{attribute 'reflection'}
{attribute 'hide_all_locals'}
FUNCTION_BLOCK Mover IMPLEMENTS iMover;

VAR_INPUT
	
	MotionParameters		: MotionParameters_typ;		// Motion parameters used by internal motion function blocks
	SourceInstancePath		: STRING	:= 'Direct access';					// Used internally to temporarily store the source of a Mover method call for logging purposes. Don't read or write

END_VAR
VAR_OUTPUT
	
	Ready			: BOOL;			// Mover is enabled and ready to accept motion commands
	Busy			: BOOL;			// Mover is processing a command or changing state
	
	Error			: BOOL;			// error is currently active
	ErrorID			: UDINT;		// errorID of the active error
	ErrorOrigin		: STRING;		// error source, in case of errored internal function block
	
	InGroup			: BOOL;			// Mover is currently grouped for CA
	IdentInGroup	: UDINT;		// IDX within group, for knowing which movers are adjacent
	
	AxisReference	: AXIS_REF;		// Motion link variable. Left as output so the link can be made directly, and accessed by external code
	
	TrackInfo		: TrackInfo;	// Track information as read from MC_ReadTrackPositions

END_VAR
VAR

	{attribute 'instance-path'}
	{attribute 'noinit'}
	{attribute 'hide'}
	InstancePath		: STRING;	// instance naming, for diagnostics purposes
	
	internalEnable		: BOOL;		// moves the axis from Disabled to Standstill, adds Axis to CA group, and triggers M1 Detection if configured
	internalDisable		: BOOL;		// moves the axis from Standstill to Disabled, removes Axis from CA Group
	
	internalCurrentMoveType			: MoverCommandType_enum;	// Most recent move command type
	internalReissue					: BOOL;						// reissue last command flag alows summing of all reissue commands per-scan
	
	internalCurrentDestPosition		: LREAL;						// Track position of the current motion destination;
	internalCurrentDestObjective	: STRING;						// Instance path of the current destination objective
	internalCurrentDestStation		: REFERENCE TO Station;			// Reference to a destination station, if that is the current movetype
	internalCurrentDestMultiStation	: REFERENCE TO MultiStation;	// Reference to a destination station, if that is the current movetype

	internalState			: MoverState_enum;		// Internal state variable
	internalTrackState		: TrackState;			// Internal state variable for track
	internalTrackStateDelay : TON;					// Internal timer for activate track delay
	
	internalMasterMover				: REFERENCE TO Mover;	// Internal reference to a target master mover
	internalMasterAxis				: REFERENCE TO AXIS_REF;	// Internal reference to a target master external axis
	internalGap						: LREAL;	// Gap distance to master mover during sync
	
	// Configurable Payload description	
	internalPayload			: Payload_typ;	// E.g. 0: No Product, 1: Product Loaded, 2: Product Reject. Can be modified for application
	
	// Track management
	internalTrack			: POINTER TO Track;	// Internal current track
	internalTrackIsReady	: BOOL := TRUE;			// track is ready for commands (off when .ActivateTrack is working)
	internalActivatingTrack : POINTER TO Track;	// while NOT .internalTrackIsReady the in-transition-to track is held here
	internalActivateTrackFlag	: BOOL;				// activate track requested
	
	// Internal function blocks	
	fbPower					: MC_Power;
	fbReset					: MC_Reset;
	fbStop					: MC_Stop;
	
	fbHaltCA				: MC_HaltCA;

	fbMoveAbsCA				: ARRAY[0..1] OF MC_MoveAbsoluteCA;
	fbAddToGroup			: MC_AddAxisToGroup;
	fbRemoveFromGroup		: MC_RemoveAxisFromGroup;
	
	fbGearInPosAxisCA		: ARRAY[0..1] OF MC_GearInPosCA;
	fbGearInPosMoverCA		: ARRAY[0..1] OF MC_GearInPosCA;
	
	fbGroupStatus			: MC_GroupReadStatus;
	fbGroupEnable			: MC_GroupEnable;
	fbGroupReset			: MC_GroupReset;
	fbGroupStop				: MC_GroupStop;
	
	fbReadStatus			: MC_ReadStatus;
	fbMoveRelCA				: ARRAY[0..1] OF MC_MoveRelativeCA;
	
	fbActivateTrack			: MC_ActivateTrack;
	fbReadTrackPositions	: MC_ReadTrackPositions;
	
	fbReadM1DetectMode		: ADSREAD;
	fbReadM1DetectValid		: ADSREAD;
	fbReadM1DetectActive	: ADSREAD;
	fbWriteM1Detect			: ADSWRITE;
	fbDelayM1Timer			: TON;
	IdDetectionMode			: DINT;			// 0: Standard 1: Mover1
	IsIdDetectionValid		: BOOL;			// M1 Detection has completed
	IsIdDetectionActive		: BOOL;			// M1 Detection currently underway
	
	// vars to store system time of most recent method calls, for filtering event logger
	
	lastCallCyclic		: LREAL;
	lastCallDisable		: LREAL;
	lastCallEnable		: LREAL;
	lastCallGroupStop	: LREAL;
	lastCallHalt		: LREAL;
	lastCallLogEvent	: LREAL;
	lastCallMovePos		: LREAL;
	lastCallMoveSta		: LREAL;
	lastCallMoveVel		: LREAL;
	lastCallReissue		: LREAL;
	lastCallSetAcc		: LREAL;
	lastCallSetDec		: LREAL;
	lastCallSetDir		: LREAL;
	lastCallSetJerk		: LREAL;
	lastCallSetVel		: LREAL;
	lastCallSync		: LREAL;
	
END_VAR
VAR_IN_OUT
	
	GroupReference		: AXES_GROUP_REF;
	
END_VAR

METHOD ActivateTrack : BOOL
VAR_INPUT
	Track	: REFERENCE TO Track;
END_VAR
VAR
	newCallTime			: LREAL;
END_VAR
VAR_INST
	MsgCreate			: FB_TcMessage;	
END_VAR
// active the track for this mover
// THIS ROUTINE IS NOT CHAINABLE wait for .IsTrackReady before issuing additional motion commands

// this routine only stores data and sets flags
// actual work of activating the track is done in .CyclicTrack()
// to enable this to be called on every scan, a check is made here for not busy as MC_ActivateTrack does not handle multiple calls efficently
// .CyclicTrack() monitors for a falling edge on internalActivateTrack before allowing another command
// this functionality mimics motion library commands such as MC_MoveAbsolute
internalActivateTrackFlag := TRUE;
IF (internalTrackState = TrackState.WAIT_FOR_COMMAND) THEN
	internalActivatingTrack := ADR(Track);
	internalTrackIsReady := FALSE;
	
	newCallTime		:= ULINT_TO_LREAL(F_GetSystemTime())/1E7;
	
	IF ( newCallTime - lastCallMoveSta ) > 1 THEN
		MsgCreate.CreateEx( TC_EVENTS.XtsBaseEventClass.MoverActivateTrack,0 );
		MsgCreate.ipArguments.Clear().AddString(THIS^.InstancePath).AddInt(internalActivatingTrack^.Id).AddString(THIS^.SourceInstancePath).AddString(Track.InstancePath);
		MsgCreate.Send(0);
	END_IF
	
	lastCallMovePos		:= newCallTime;
END_IF;
END_METHOD

{attribute 'monitoring' := 'call'}
PROPERTY CurrentDestinationPosition : LREAL
GET

CurrentDestinationPosition		:= internalCurrentDestPosition;
END_GET
END_PROPERTY

{attribute 'monitoring' := 'call'}
PROPERTY CurrentMoveType : MoverCommandType_enum
GET
VAR
	MoverCurrentMoveType: MoverCommandType_enum;
END_VAR

CurrentMoveType		:= internalCurrentMoveType;
END_GET
END_PROPERTY

{attribute 'monitoring' := 'call'}
PROPERTY CurrentObjective : String
GET

CurrentObjective		:= internalCurrentDestObjective;
END_GET
END_PROPERTY

PROPERTY CurrentTrack : POINTER TO Track
GET
CurrentTrack := internalTrack;
END_GET
END_PROPERTY

METHOD Cyclic : iMover
VAR_IN_OUT
	GroupReference		: AXES_GROUP_REF;
END_VAR





// cleans motion parameters, removing possible negatives. Upper bounds are capped by the axis parameters
MotionParameters.Acceleration	:= LIMIT( 0, MotionParameters.Acceleration, 1E300 );
MotionParameters.Deceleration	:= LIMIT( 0, MotionParameters.Deceleration, 1E300 );
MotionParameters.Jerk			:= LIMIT( 0, MotionParameters.Jerk, 1E300 );
MotionParameters.Velocity		:= LIMIT( 0, MotionParameters.Velocity, 1E300 );






CASE internalState OF
	MV_IDLE:	// ------------------------------------------------------- idle state
	
		Ready	:= FALSE;
		Busy	:= FALSE;

		fbMoveAbsCA[0].Execute	:= FALSE;
		fbMoveAbsCA[1].Execute	:= FALSE;
		fbMoveRelCA[0].Execute	:= FALSE;
		fbMoveRelCA[1].Execute	:= FALSE;
		
		internalDisable			:= FALSE;
		IF internalEnable THEN
			internalEnable		:= FALSE;
			internalState		:= MV_RESET;
		END_IF
		
	MV_RESET: // ------------------------------------------------------- axis is resetting
	
		Ready	:= FALSE;
		Busy	:= TRUE;
		Error	:= FALSE;
		ErrorID	:= 0;
		
		fbReset.Execute			:= TRUE;
		
		IF fbReset.Done THEN
			fbReset.Execute		:= FALSE;
			internalState		:= MV_M1_READMODE;
		ELSIF fbReset.Error THEN
			ErrorID				:= fbReset.ErrorID;
			ErrorOrigin			:= CONCAT( InstancePath, '.fbReset' );
			internalState		:= MV_ERROR;		
		END_IF
		
	MV_M1_READMODE: // ------------------------------------------------------- begin checking for M1 detection mode setting
	
		Ready	:= FALSE;
		Busy	:= TRUE;
		Error	:= FALSE;
		ErrorID	:= 0;
		
		// todo: values may change. see issue #25 for update
		fbReadM1DetectMode.NETID		:= '';
		fbReadM1DetectMode.PORT			:= 351;
		fbReadM1DetectMode.IDXGRP		:= GVL.pXtsProcessingUnit;
		fbReadM1DetectMode.IDXOFFS		:= 16#03080246;
		fbReadM1DetectMode.LEN			:= SIZEOF( IdDetectionMode );
		fbReadM1DetectMode.DESTADDR		:= ADR( IdDetectionMode );
		fbReadM1DetectMode.READ			:= TRUE;
		
		internalState	:= MV_M1_EVALMODE;
		
	MV_M1_EVALMODE: // ------------------------------------------------------- Determine detection mode setting
	
		Ready	:= FALSE;
		Busy	:= TRUE;
		Error	:= FALSE;
		ErrorID	:= 0;
	
		fbReadM1DetectMode.READ		:= FALSE;
		
		CASE IdDetectionMode OF
			0:	internalState		:= MV_ENABLING;			// Mover 1 functionality is not configured, skip ahead to enabling the mover
			1:	internalState		:= MV_M1_READSTATUS;	// Mover 1 functionality is configured, read detection status
		END_CASE
	
	MV_M1_READSTATUS: // ------------------------------------------------------- Determine current M1 Detection Status
	
		Ready	:= FALSE;
		Busy	:= TRUE;
		Error	:= FALSE;
		ErrorID	:= 0;
		
		fbWriteM1Detect.WRITE			:= FALSE;
		
		fbReadM1DetectValid.NETID		:= '';
		fbReadM1DetectValid.PORT		:= 351;
		fbReadM1DetectValid.IDXGRP		:= GVL.pXtsProcessingUnit;
		fbReadM1DetectValid.IDXOFFS		:= 16#03080251;
		fbReadM1DetectValid.LEN			:= SIZEOF( IsIdDetectionValid );
		fbReadM1DetectValid.DESTADDR	:= ADR( IsIdDetectionValid );
		fbReadM1DetectValid.READ		:= TRUE;
		
		fbReadM1DetectActive.NETID		:= '';
		fbReadM1DetectActive.PORT		:= 351;
		fbReadM1DetectActive.IDXGRP		:= GVL.pXtsProcessingUnit;
		fbReadM1DetectActive.IDXOFFS	:= 16#03080268;
		fbReadM1DetectActive.LEN		:= SIZEOF( IsIdDetectionActive );
		fbReadM1DetectActive.DESTADDR	:= ADR( IsIdDetectionActive );
		fbReadM1DetectActive.READ		:= TRUE;
		
		internalState	:= MV_M1_EVALSTATUS;
		
	MV_M1_EVALSTATUS:	// ------------------------------------------------------- Determine to activate M1 Detect or ignore
	
		Ready	:= FALSE;
		Busy	:= TRUE;
		Error	:= FALSE;
		ErrorID	:= 0;
	
		fbReadM1DetectValid.READ		:= FALSE;
		fbReadM1DetectActive.READ		:= FALSE;
		
		IF IsIdDetectionActive THEN
			internalState		:= MV_M1_READSTATUS;	// M1 Detection is underway, but we need to wait until it completes
		ELSIF IsIdDetectionValid THEN
			internalState		:= MV_ENABLING;			// M1 Detection complete, ready to enable this mover
		ELSE
			internalState		:= MV_M1_DETECT;		// M1 Detection hasn't been started yet. So start it!
		END_IF
 
	MV_M1_DETECT:	// ------------------------------------------------------- Begin M1 Detection
	
		Ready	:= FALSE;
		Busy	:= TRUE;
		Error	:= FALSE;
		ErrorID	:= 0;
		
		fbWriteM1Detect.NETID			:= '';
		fbWriteM1Detect.PORT			:= 351;
		fbWriteM1Detect.IDXGRP			:= GVL.pXtsProcessingUnit;
		fbWriteM1Detect.IDXOFFS			:= 16#03080250;
		fbWriteM1Detect.WRITE			:= TRUE;
		
		internalState	:= MV_M1_DELAY;	// go back to Read M1 Detect status to confirm it has completed
		
	MV_M1_DELAY:	// ------------------------------------------------------ delay to allow M1 Detect Completion
	
		Ready	:= FALSE;
		Busy	:= TRUE;
		Error	:= FALSE;
		ErrorID	:= 0;
		
		fbDelayM1Timer( IN := TRUE, PT := T#500MS );
		
		IF fbDelayM1Timer.Q THEN
			fbDelayM1Timer( IN := FALSE );
			internalState	:= MV_M1_READSTATUS;
		END_IF
			
	MV_ENABLING: // ------------------------------------------------------- axis is enabling
	
		Ready	:= FALSE;
		Busy	:= TRUE;
		Error	:= FALSE;
		ErrorID	:= 0;
		
		fbPower.Enable					:= TRUE;
		fbPower.Enable_Positive			:= TRUE;
		fbPower.Enable_Negative			:= TRUE;
		fbPower.BufferMode				:= MC_Aborting;
		fbPower.Override				:= 100;
		
		IF fbPower.Status THEN
			internalState				:= MV_ADDTOGROUP;
		ELSIF fbPower.Error THEN
			ErrorID						:= fbPower.ErrorID;
			ErrorOrigin					:= CONCAT( InstancePath, '.fbPower' );
			internalState				:= MV_ERROR;
		END_IF
		
	MV_ADDTOGROUP: // ------------------------------------------------------- axis is adding to a group
	
		Ready	:= FALSE;
		Busy	:= TRUE;
		Error	:= FALSE;
		ErrorID	:= 0;
		
		fbAddToGroup.Execute			:= TRUE;
		fbAddToGroup.IdentInGroup		:= UDINT_TO_IDENTINGROUP( AxisReference.NcToPlc.AxisId - 1 );
		
		IF fbAddToGroup.Done THEN
			InGroup						:= TRUE;
			IdentInGroup				:= AxisReference.NcToPlc.AxisId - 1;
			fbAddToGroup.Execute		:= FALSE;
			internalState				:= MV_READGROUPSTATUS;
		ELSIF fbAddToGroup.Error THEN
			ErrorID						:= fbAddToGroup.ErrorId;
			ErrorOrigin					:= CONCAT( InstancePath, '.fbAddToGroup' );
			internalState				:= MV_ERROR;
		END_IF
		
	MV_READGROUPSTATUS: // ------------------------------------------------------- check the status of the group
	
		Ready	:= FALSE;
		Busy	:= TRUE;
		Error	:= FALSE;
		ErrorID	:= 0;
		
		fbGroupStatus.Enable			:= TRUE;
		
		fbGroupStatus( AxesGroup := GroupReference );	// get current information
		
		IF fbGroupStatus.Valid AND fbGroupStatus.GroupErrorStop THEN
			fbGroupReset.Execute		:= TRUE;
		ELSIF fbGroupStatus.Valid AND fbGroupStatus.GroupDisabled THEN
			fbGroupReset.Execute		:= FALSE;
			internalState				:= MV_ENABLEGROUP;
		ELSIF fbGroupStatus.Valid AND ( fbGroupStatus.GroupStandby OR fbGroupStatus.GroupMoving ) THEN
			fbGroupReset.Execute		:= FALSE;
			internalState				:= MV_RUN;
		END_IF
		
		IF fbGroupStatus.Error THEN
			ErrorID						:= fbGroupStatus.ErrorId;
			ErrorOrigin					:= CONCAT( InstancePath, '.fbGroupStatus' );
			internalState				:= MV_ERROR;
		ELSIF fbGroupReset.Error THEN
			ErrorID						:= fbGroupStatus.ErrorId;
			ErrorOrigin					:= CONCAT( InstancePath, '.fbGroupReset' );
			internalState				:= MV_ERROR;
		END_IF
		
	
	MV_ENABLEGROUP: // ------------------------------------------------------- enable the group
	
		Ready	:= FALSE;
		Busy	:= TRUE;
		Error	:= FALSE;
		ErrorID	:= 0;
		
		fbGroupEnable.Execute			:= TRUE;
		
		IF fbGroupEnable.Done THEN
			fbGroupEnable.Execute		:= FALSE;
			internalState				:= MV_RUN;
		ELSIF fbGroupEnable.Error THEN
			ErrorID						:= fbGroupEnable.ErrorId;
			ErrorOrigin					:= CONCAT( InstancePath, '.fbGroupEnable' );
			internalState				:= MV_ERROR;
		END_IF
		
	MV_RUN: // ------------------------------------------------------- mover enabled, ready
	
		Ready	:= TRUE;
		IF NOT fbMoveAbsCA[0].busy AND NOT fbMoveAbsCA[1].Busy AND NOT fbMoveRelCA[0].Busy AND NOT fbMoveRelCA[1].Busy THEN 
			Busy	:= FALSE;
		ELSE
			Busy 	:= TRUE;
		END_IF
		Error	:= FALSE;
		ErrorID	:= 0;
		
		internalEnable			:= FALSE;		
		IF internalDisable THEN
			internalDisable		:= FALSE;
			internalState		:= MV_BEGIN_HALTING;
			
		// Reset all commands issued by method calls
		ELSIF fbMoveAbsCA[0].Busy OR fbMoveAbsCA[0].CommandAborted THEN // OR fbMoveAbs.CommandAborted THEN
			fbMoveAbsCA[0].Execute		:= FALSE;
		ELSIF fbMoveAbsCA[1].Busy OR fbMoveAbsCA[1].CommandAborted THEN
			fbMoveAbsCA[1].Execute		:= FALSE;			
		ELSIF fbAddToGroup.Done THEN
			fbAddToGroup.Execute		:= FALSE;
		ELSIF fbMoveRelCA[0].Busy OR fbMoveRelCA[0].CommandAborted THEN
			fbMoveRelCA[0].Execute		:= FALSE;
		ELSIF fbMoveRelCA[1].Busy OR fbMoveRelCA[1].CommandAborted THEN
			fbMoveRelCA[1].Execute		:= FALSE;
		ELSIF fbGearInPosMoverCA[0].Busy OR fbGearInPosMoverCA[0].CommandAborted THEN
			fbGearInPosMoverCA[0].Execute	:= FALSE;
		ELSIF fbGearInPosMoverCA[1].Busy OR fbGearInPosMoverCA[1].CommandAborted THEN
			fbGearInPosMoverCA[1].Execute	:= FALSE;
		ELSIF fbGearInPosAxisCA[0].Busy OR fbGearInPosAxisCA[0].CommandAborted THEN
			fbGearInPosAxisCA[0].Execute	:= FALSE;
		ELSIF fbGearInPosAxisCA[1].Busy OR fbGearInPosAxisCA[1].CommandAborted THEN
			fbGearInPosAxisCA[1].Execute	:= FALSE;
		ELSIF fbHaltCA.Busy OR fbHaltCA.CommandAborted OR fbHaltCA.Done THEN
			fbHaltCA.Execute			:= FALSE;
		// This is different than the other similar cases, since a Stop command should prevent other commands from overriding it, thus
		// the Execute needs to remain High until the command has fully completed.
		ELSIF fbGroupStop.Done THEN
			fbGroupStop.Execute			:= FALSE;
		END_IF;
		
		THIS^.CyclicTrack();
		
		IF (internalReissue) THEN
			THIS^.SourceInstancePath	:= 'ReissueCommand';

			CASE internalCurrentMoveType OF
				MOVETYPE_NONE:
					// No current command to reissue	
				MOVETYPE_POSITION:
					THIS^.MoveToPosition( internalCurrentDestPosition );
				MOVETYPE_STATION:
					THIS^.MoveToStation( internalCurrentDestStation );
				MOVETYPE_MULTISTATION:
					THIS^.MoveToStation( internalCurrentDestStation );
				MOVETYPE_VELOCITY:
					THIS^.MoveVelocity( MotionParameters.Velocity );
				MOVETYPE_SYNC_MOVER:
					THIS^.SyncToMover( internalMasterMover, internalGap );
				MOVETYPE_SYNC_AXIS:
					// This command should perhaps not be compatible with Reissue command
			END_CASE
			internalReissue := FALSE;
		END_IF

		// And catch all internal function block errors
		IF fbMoveAbsCA[0].Error THEN
			ErrorID					:= fbMoveAbsCA[0].ErrorID;
			ErrorOrigin				:= CONCAT( InstancePath, '.fbMoveAbs[0]' );
			internalState			:= MV_ERROR;
		ELSIF fbMoveAbsCA[1].Error THEN
			ErrorID					:= fbMoveAbsCA[1].ErrorId;
			ErrorOrigin				:= CONCAT( InstancePath, '.fbMoveAbs[1]' );
			internalState			:= MV_ERROR;
		ELSIF fbAddToGroup.Error THEN
			ErrorID					:= fbAddToGroup.ErrorID;
			ErrorOrigin				:= CONCAT( InstancePath, '.fbAddToGroup' );
			internalState			:= MV_ERROR;
		ELSIF fbGroupStop.Error THEN
			ErrorID					:= fbGroupStop.ErrorId;
			ErrorOrigin				:= CONCAT( InstancePath, '.fbGroupStop' );
			internalState			:= MV_ERROR;
		ELSIF fbMoveRelCA[0].Error THEN
			ErrorID					:= fbMoveRelCA[0].ErrorID;
			ErrorOrigin 			:= CONCAT ( InstancePath, '.fbMoveRelCA[0]');
			internalState			:= MV_ERROR;
		ELSIF fbMoveRelCA[1].Error THEN
			ErrorID					:= fbMoveRelCA[1].ErrorID;
			ErrorOrigin 			:= CONCAT ( InstancePath, '.fbMoveRelCA[1]');
			internalState			:= MV_ERROR;
		ELSIF fbReadStatus.Valid AND fbReadStatus.ErrorStop THEN
			ErrorID					:= fbReadStatus.Status.ErrorID;
			ErrorOrigin				:= CONCAT( InstancePath, '.fbReadStatus' );
			internalState			:= MV_ERROR;
		ELSIF fbGearInPosMoverCA[0].Error THEN
			ErrorID					:= fbGearInPosMoverCA[0].ErrorId;
			ErrorOrigin				:= CONCAT( InstancePath, '.fbGearInPosMoverCA[0]');
			internalState			:= MV_ERROR;
		ELSIF fbGearInPosMoverCA[1].Error THEN
			ErrorID					:= fbGearInPosMoverCA[1].ErrorId;
			ErrorOrigin				:= CONCAT( InstancePath, '.fbGearInPosMoverCA[1]');
			internalState			:= MV_ERROR;
		ELSIF fbGearInPosAxisCA[0].Error THEN
			ErrorID					:= fbGearInPosAxisCA[0].ErrorId;
			ErrorOrigin				:= CONCAT( InstancePath, '.fbGearInPosAxisCA[0]');
			internalState			:= MV_ERROR;
		ELSIF fbGearInPosAxisCA[1].Error THEN
			ErrorID					:= fbGearInPosAxisCA[1].ErrorId;
			ErrorOrigin				:= CONCAT( InstancePath, '.fbGearInPosAxisCA[1]');
			internalState			:= MV_ERROR;			
		ELSIF fbActivateTrack.Error THEN
			ErrorID					:= fbActivateTrack.ErrorId;
			ErrorOrigin				:= CONCAT( InstancePath, '.fbActivateTrack');
			internalState			:= MV_ERROR;
		END_IF
		
	MV_BEGIN_HALTING:	// --------------------------------------------------- begin stopping process
	
		Ready	:= FALSE;
		Busy	:= TRUE;
		Error	:= FALSE;
		ErrorID	:= 0;
		
		// Kill any active motion commands
		fbMoveRelCA[0].Execute		:= FALSE;
		fbMoveRelCA[1].Execute		:= FALSE;
		fbMoveAbsCA[0].Execute		:= FALSE;
		fbMoveAbsCA[1].Execute		:= FALSE;
				
		IF fbReadStatus.ErrorStop = FALSE THEN
			fbHaltCA.Execute		:= TRUE;
			//fbHaltCA.Deceleration	:= MotionParameters.Deceleration;
			//fbHaltCA.Jerk			:= MotionParameters.Jerk;
		ELSE
			internalState			:= MV_REMOVEFROMGROUP;
		END_IF;
		
		IF fbHaltCA.Active OR fbHaltCA.Done THEN
			internalState			:= MV_HALTING;
		ELSIF fbHaltCA.Error THEN
			ErrorID					:= fbHaltCA.ErrorID;
			ErrorOrigin				:= CONCAT( InstancePath, '.fbHalt' );
			internalState			:= MV_ERROR;				
		END_IF	
		
	MV_HALTING:	// ------------------------------------------------------- mover disabling
	
		Ready	:= FALSE;
		Busy	:= TRUE;
		Error	:= FALSE;
		ErrorID	:= 0;

		// Wait for the stopping action to complete
		IF fbHaltCA.Done THEN
			fbHaltCA.Execute		:= FALSE;
			internalState			:= MV_REMOVEFROMGROUP;
		ELSIF fbHaltCA.Error THEN
			ErrorID					:= fbStop.ErrorID;
			ErrorOrigin				:= CONCAT( InstancePath, '.fbHalt' );
			internalState			:= MV_ERROR;
		END_IF	
		
	MV_REMOVEFROMGROUP:	// ---------------------------------------------------- remove mover from CA group
	
		Ready	:= FALSE;
		Busy	:= TRUE;
		Error	:= FALSE;
		ErrorID	:= 0;
		
		fbRemoveFromGroup.Execute			:= TRUE;
		fbRemoveFromGroup.IdentInGroup		:= UDINT_TO_IDENTINGROUP( IdentInGroup );
		
		IF fbRemoveFromGroup.Done THEN
			fbRemoveFromGroup.Execute		:= FALSE;
			internalState					:= MV_DISABLING;
		END_IF
		


	MV_DISABLING:	// ----------------------------------------------------- start the disabling process

		Ready	:= FALSE;
		Busy	:= TRUE;
		Error	:= FALSE;
		ErrorID	:= 0;
		
		fbPower.Enable				:= FALSE;
		fbPower.Enable_Positive		:= FALSE;
		fbPower.Enable_Negative		:= FALSE;
		fbPower.BufferMode			:= MC_Aborting;
		fbPower.Override			:= 100;
			
		IF fbPower.Status = FALSE THEN
			internalState			:= MV_IDLE;
		ELSIF fbPower.Error THEN
			ErrorID					:= fbPower.ErrorID;
			ErrorOrigin				:= CONCAT( InstancePath, '.fbPower' );
			internalState			:= MV_ERROR;
		END_IF		
	
	MV_ERROR: // ------------------------------------------------------- mover in error state
	
		Ready	:= FALSE;
		Busy	:= FALSE;
		Error	:= TRUE;
		
		internalEnable			:= FALSE;		
		IF internalDisable THEN
			internalDisable		:= FALSE;
			internalState		:= MV_REMOVEFROMGROUP;
			ErrorOrigin			:= '';
		END_IF
		
END_CASE

fbPower( Axis := AxisReference );
fbReset( Axis := AxisReference );
fbStop( Axis := AxisReference );

fbHaltCA( Axis := AxisReference );
//fbDisable( Axis := AxisRef );
//fbExternEnable( Axis := AxisRef );

fbAddToGroup( AxesGroup := GroupReference, Axis := AxisReference );
fbRemoveFromGroup( AxesGroup := GroupReference );

fbGroupStatus( AxesGroup := GroupReference );
fbGroupEnable( AxesGroup := GroupReference );
fbGroupReset( AxesGroup := GroupReference );
fbGroupStop( AxesGroup := GroupReference );

fbMoveAbsCA[0]( Axis := AxisReference );
fbMoveAbsCA[1]( Axis := AxisReference );
fbReadStatus( Enable := TRUE, Axis := AxisReference );
fbMoveRelCA[0] ( Axis := AxisReference );
fbMoveRelCA[1] ( Axis := AxisReference );

fbGearInPosMoverCA[0]( Master := internalMasterMover.AxisReference, Slave := THIS^.AxisReference );
fbGearInPosMoverCA[1]( Master := internalMasterMover.AxisReference, Slave := THIS^.AxisReference );

fbGearInPosAxisCA[0]( Master := internalMasterAxis, Slave := THIS^.AxisReference );
fbGearInPosAxisCA[1]( Master := internalMasterAxis, Slave := THIS^.AxisReference );

fbReadM1DetectMode();
fbReadM1DetectValid();
fbReadM1DetectActive();
fbWriteM1Detect();

// track management
fbActivateTrack(Axis := AxisReference);
fbReadTrackPositions(Axis := AxisReference);
END_METHOD

METHOD CyclicTrack : BOOL
VAR
END_VAR
VAR_INST
	MsgCreate			: FB_TcMessage;	
END_VAR
// called by .Cyclic() to handle the MC_ActivateTrack call's required state machine
// this is only called while the mover is in the RUN state within .Cyclic() by design
// calling the track management functions on disabled or errored movers that are not
// assigned to a group just causes the track management functions to throw more errors

CASE internalTrackState OF
	// wait for command
	TrackState.WAIT_FOR_COMMAND:
		IF (internalActivateTrackFlag) THEN
			// unregister mover from current track (logical tracking)
			IF (internalTrack <> 0) THEN
				internalTrack^.UnregisterMover(THIS^);
			END_IF;

			// set flags
			internalTrack := ADR(ErrorTrack);
			internalTrackIsReady := FALSE;

			// advance state
			internalTrackState := TrackState.SETUP_FUNCTION;
		END_IF
		
	// setup and call the function
	TrackState.SETUP_FUNCTION:
		fbActivateTrack.TrackId := internalActivatingTrack^.OTCID;
		fbActivateTrack.Execute := TRUE;
		IF (fbActivateTrack.Busy) THEN
			fbActivateTrack.Execute := FALSE;
			internalTrackState := TrackState.MONITOR_RESPONSE;
		END_IF
	
	// monitor response	
	TrackState.MONITOR_RESPONSE:
		IF (fbActivateTrack.Error) THEN
			internalTrackState := TrackState.ERROR;
		ELSIF (fbActivateTrack.Done) THEN
			internalTrackState := TrackState.REQUIRED_DELAY;
		END_IF;
	
	// required delay
	// the FB has returned .Done but the change has not yet propigated to the NC
	TrackState.REQUIRED_DELAY:
		internalTrackStateDelay.IN := TRUE;
		IF (internalTrackStateDelay.Q) THEN
			internalTrackStateDelay.IN := FALSE;
			internalTrackState := TrackState.CLEAN_UP;
		END_IF;
	
	// clean up flags
	TrackState.CLEAN_UP:
		internalTrack := internalActivatingTrack;
		internalActivatingTrack := ADR(ErrorTrack);
		internalTrackIsReady := TRUE;
		MsgCreate.CreateEx( TC_EVENTS.XtsBaseEventClass.MoverActivateTrackComplete, 0);
		MsgCreate.ipArguments.Clear().AddString(THIS^.InstancePath).AddInt(THIS^.CurrentTrack^.Id);
		MsgCreate.Send(0);
		internalTrackState := TrackState.WAIT_END;
		
	TrackState.ERROR:
		// reset execute
		fbActivateTrack.Execute := FALSE;
		// GVL.ERROR_TRACK is intentionally left in place
		// internalTrackIsReady is left at false
		// error is recorded in Cyclic()
		internalTrackState := TrackState.WAIT_END;
		
	TrackState.WAIT_END: 
		// falling edge detection for internalActivateTrackFlag
		IF (NOT internalActivateTrackFlag) THEN
			// register mover
			internalTrack^.RegisterMover(THIS^);
			internalTrackState := TrackState.WAIT_FOR_COMMAND;	
		END_IF
		internalActivateTrackFlag := FALSE;

END_CASE

// read back track information
IF (internalTrackIsReady) THEN
	// track info should be stable, call the block
	fbReadTrackPositions.Enable := TRUE;
	// copy data when ready
	IF (fbReadTrackPositions.Valid) THEN
		TrackInfo.TrackPosition := LMOD(fbReadTrackPositions.TrackPosition, GVL.TRACK_LENGTH);
		TrackInfo.PartPosition := LMOD(fbReadTrackPositions.PartPosition, GVL.TRACK_LENGTH);
		TrackInfo.TrackId := fbReadTrackPositions.TrackId;
		TrackInfo.PartId := fbReadTrackPositions.PartId;
	END_IF
ELSE
	// don't call function block to allow it to reset
	fbReadTrackPositions.Enable := FALSE;
END_IF


// a delay is required after MC_ActivateTrack returns .Done
internalTrackStateDelay(PT := T#10MS);
END_METHOD

METHOD Disable : iMover
VAR_INPUT
END_VAR
VAR
END_VAR
VAR_INST
	MsgCreate	: FB_TcMessage;	
END_VAR

IF internalState = MV_RUN OR internalState = MV_ERROR THEN

	// Sets an internal flag to advance the state machine
	internalDisable		:= TRUE;
	
	MsgCreate.CreateEx( TC_EVENTS.XtsBaseEventClass.MoverDisable,0 );
	MsgCreate.ipArguments.Clear().AddString(THIS^.InstancePath).AddString(THIS^.SourceInstancePath);
	MsgCreate.Send(0);	
END_IF

THIS^.SourceInstancePath	:= 'Direct access';

Disable		:= THIS^;
END_METHOD

METHOD Enable : iMover
VAR_INPUT
END_VAR
VAR
END_VAR
VAR_INST
	MsgCreate	: FB_TcMessage;	
END_VAR

IF internalState = MV_IDLE THEN

	// Sets an internal flag to advance the state machine
	internalEnable		:= TRUE;
	
	MsgCreate.CreateEx( TC_EVENTS.XtsBaseEventClass.MoverEnable,0 );
	MsgCreate.ipArguments.Clear().AddString(THIS^.InstancePath).AddString(THIS^.SourceInstancePath);
	MsgCreate.Send(0);

END_IF;

THIS^.SourceInstancePath	:= 'Direct access';

Enable := THIS^;
END_METHOD

METHOD GroupStop : iMover
VAR_INPUT
END_VAR
VAR
	newCallTime	: LREAL;
END_VAR
VAR_INST
	MsgCreate	: FB_TcMessage;	
END_VAR


IF NOT( Ready ) THEN	// if the mover is not ready & able to accept a GroupHalt Command

	internalState	:= MV_ERROR;
	ErrorID			:= 19201;

ELSE	// otherwise execute the command
	
	// grab a timestamp of the command
	newCallTime		:= ULINT_TO_LREAL(F_GetSystemTime())/1E7;
	
	fbGroupStop.Execute			:= TRUE;
	fbGroupStop.Deceleration	:= MotionParameters.Deceleration;
	fbGroupStop.Jerk			:= MotionParameters.Jerk;
	
	memset( ADR( internalCurrentDestObjective ), 0, SIZEOF( internalCurrentDestObjective ));
	internalCurrentMoveType		:= MoverCommandType_enum.MOVETYPE_NONE;
	
END_IF

IF ( newCallTime - lastCallGroupStop ) > 1 THEN
	MsgCreate.CreateEx( TC_EVENTS.XtsBaseEventClass.MoverGroupStop,0 );
	MsgCreate.ipArguments.Clear().AddString(THIS^.InstancePath).AddString(THIS^.SourceInstancePath);
	MsgCreate.Send(0);
END_IF

THIS^.SourceInstancePath	:= 'Direct access';

lastCallGroupStop	:= newCallTime;

GroupStop		:= THIS^;
END_METHOD

METHOD Halt : iMover
VAR_INPUT
END_VAR
VAR
	newCallTime: LREAL;
END_VAR
VAR_INST
	MsgCreate: FB_TcMessage;	
END_VAR

IF NOT( Ready ) THEN
	
	internalState	:= MV_ERROR;
	ErrorID			:= 19201;
	
ELSIF fbHaltCA.Busy THEN	

	newCallTime		:= ULINT_TO_LREAL(F_GetSystemTime())/1E7;
	
	// oddly, MC_HaltCA does not include an option for BufferMode
	// so do nothing
	
ELSE
	
	newCallTime		:= ULINT_TO_LREAL(F_GetSystemTime())/1E7;
	
	fbHaltCA.Execute		:= TRUE;
	fbHaltCA.Deceleration	:= MotionParameters.Deceleration;
	fbHaltCA.Jerk			:= MotionParameters.Jerk;
	
	fbHaltCA( Axis := AxisReference );
	
END_IF

internalCurrentMoveType		:= MOVETYPE_NONE;
internalCurrentDestPosition	:= 1E300;

memset( ADR( internalCurrentDestObjective), 0, SIZEOF( internalCurrentDestObjective ));
internalCurrentDestStation	REF= 0;

IF ( newCallTime - lastCallHalt ) > 1 THEN
	MsgCreate.CreateEx( TC_EVENTS.XtsBaseEventClass.MoverHalt,0);
	MsgCreate.ipArguments.Clear().AddString(THIS^.InstancePath).AddString(THIS^.SourceInstancePath).AddLReal(MotionParameters.Deceleration);
	MsgCreate.Send(0);
END_IF

THIS^.SourceInstancePath	:= 'Direct access';

lastCallHalt		:= newCallTIme;

Halt	:= THIS^;
END_METHOD

{attribute 'monitoring' := 'call'}
PROPERTY IsSyncedToAxis : BOOL
GET


IsSyncedToAxis		:= fbGearInPosAxisCA[0].InSync OR fbGearInPosAxisCA[1].InSync;
END_GET
END_PROPERTY

{attribute 'monitoring' := 'call'}
PROPERTY IsSyncedToMover : BOOL
GET


IsSyncedToMover		:= fbGearInPosMoverCA[0].InSync OR fbGearInPosMoverCA[1].InSync;
END_GET
END_PROPERTY

PROPERTY IsTrackReady : BOOL
GET
IsTrackReady := internalTrackIsReady;
END_GET
END_PROPERTY

METHOD LogUserEvent : iMover
VAR_INPUT
	String1	: STRING;	// First content section of user-event message
	String2 : STRING;	// Second content section of user-event message
	String3 : STRING;	// Third content section of user-event message
END_VAR
VAR
END_VAR
VAR_INST
	MsgCreate: FB_TcMessage;	
END_VAR



MsgCreate.CreateEx( TC_EVENTS.XtsBaseEventClass.UserEvent, 0 );
MsgCreate.ipArguments.Clear().AddString(String1).AddString(String2).AddString(String3);
MsgCreate.Send(0);

LogUserEvent	:= THIS^;
END_METHOD

PROPERTY MasterMover : Reference To Mover
GET


IF THIS^.internalCurrentMoveType = MOVETYPE_SYNC_MOVER THEN
	MasterMover		REF= internalMasterMover;
ELSE
	MasterMover		REF= 0;
END_IF
END_GET
END_PROPERTY

METHOD MoveToMultiStation : iMover
VAR_INPUT
	DestinationStation	: REFERENCE TO MultiStation;	
END_VAR
VAR
	newCallTime			: LREAL;
END_VAR
VAR_INST
	MsgCreate			: FB_TcMessage;	
END_VAR
IF NOT( Ready ) AND NOT(__ISVALIDREF( DestinationStation )) THEN	// if the mover is not ready & able to accept a moveabs command...
	
	internalState	:= MV_ERROR;
	ErrorID			:= 19201;
	
ELSE	// otherwise let 'er rip
	
	newCallTime		:= ULINT_TO_LREAL(F_GetSystemTime())/1E7;
	internalReissue := FALSE;	// reissue no longer necessary
	
	IF fbMoveAbsCA[0].Busy = FALSE THEN
		
		fbMoveAbsCA[0].Jerk			:= MotionParameters.Jerk;
		fbMoveAbsCA[0].Acceleration	:= MotionParameters.Acceleration;
		fbMoveAbsCA[0].Deceleration	:= MotionParameters.Deceleration;
		fbMoveAbsCA[0].Velocity		:= MotionParameters.Velocity;
		fbMoveAbsCA[0].Direction	:= MotionParameters.Direction;
		fbMoveAbsCA[0].Options.DynamicsReferenceSystem := CurrentTrack^.OTCID;
		fbMoveAbsCA[0].Options.PositionReferenceSystem := CurrentTrack^.OTCID;
		
//		fbMoveAbsCA[0].Position		:= DestinationStation.internalPosition;
		fbMoveAbsCA[0].Position		:= DestinationStation.Station[0].Position;
		
		fbMoveAbsCA[0].BufferMode	:= mcAborting;
		fbMoveAbsCA[0].Execute		:= TRUE;
		 
		fbMoveAbsCA[0].Execute		:= TRUE;		// execute this block, and...
		fbMoveAbsCA[1].Execute		:= FALSE;		// if necessary, interrupt this one
		
		fbMoveAbsCA[0]( Axis := AxisReference );
		
	ELSIF fbMoveAbsCA[1].Busy = FALSE THEN
		
		fbMoveAbsCA[1].Jerk			:= MotionParameters.Jerk;
		fbMoveAbsCA[1].Acceleration	:= MotionParameters.Acceleration;
		fbMoveAbsCA[1].Deceleration	:= MotionParameters.Deceleration;
		fbMoveAbsCA[1].Velocity		:= MotionParameters.Velocity;
		fbMoveAbsCA[1].Direction	:= MotionParameters.Direction;
		fbMoveAbsCA[1].Options.DynamicsReferenceSystem := CurrentTrack^.OTCID;
		fbMoveAbsCA[1].Options.PositionReferenceSystem := CurrentTrack^.OTCID;
		
//		fbMoveAbsCA[1].Position		:= DestinationStation.internalPosition;
		fbMoveAbsCA[1].Position		:= DestinationStation.Station[0].Position;
		
		fbMoveAbsCA[1].BufferMode	:= mcAborting;
		fbMoveAbsCA[1].Execute		:= TRUE;
		
		fbMoveAbsCA[1].Execute		:= TRUE;		// execute this block, and...
		fbMoveAbsCA[0].Execute		:= FALSE;		// if necessary, interrupt this one

		fbMoveAbsCA[1]( Axis := AxisReference );	

	ELSE
		MsgCreate.CreateEx( TC_EVENTS.XtsBaseEventClass.MoverMoveToStationOverload,0 );
		MsgCreate.ipArguments.Clear().AddString(THIS^.InstancePath).AddString(THIS^.SourceInstancePath).AddString(DestinationStation.InstancePath);
		MsgCreate.Send(0);
		
	END_IF
	
	// Set the current destination object to the instance path of the objective, or 0 if unassigned
	internalCurrentDestPosition		:= DestinationStation.Position;
	internalCurrentDestObjective	:= SEL( __ISVALIDREF( DestinationStation ), '', DestinationStation.InstancePath );
	internalCurrentDestMultiStation	REF= DestinationStation;
	internalCurrentMoveType			:= MOVETYPE_MULTISTATION;
	
	// Register this mover with the station, so the station knows this mover is incoming
	DestinationStation.RegisterMover( THIS^ );
	
END_IF

IF ( newCallTime - lastCallMoveSta ) > 1 THEN
	MsgCreate.CreateEx( TC_EVENTS.XtsBaseEventClass.MoverMoveToStation,0 );
	MsgCreate.ipArguments.Clear().AddString(THIS^.InstancePath).AddString(THIS^.SourceInstancePath).AddString(DestinationStation.InstancePath);
	MsgCreate.Send(0);
END_IF

THIS^.SourceInstancePath	:= 'Direct access';

lastCallMoveSta		:= newCallTime;

MoveToMultiStation		:= THIS^;
END_METHOD

METHOD PUBLIC MoveToPosition : iMover
VAR_INPUT
	DestinationPosition		: LREAL;	// position on track for a shuttle to move towards
END_VAR
VAR
	newCallTime		: LREAL;
END_VAR
VAR_INST
	MsgCreate		: FB_TcMessage;	
END_VAR

IF NOT( Ready ) THEN	// if the mover is not ready & able to accept a moveabs command...
	
	internalState	:= MV_ERROR;
	ErrorID			:= 19201;
	
ELSE	// otherwise let 'er rip
	
	newCallTime		:= ULINT_TO_LREAL(F_GetSystemTime())/1E7;
	internalReissue := FALSE;	// reissue no longer necessary
	
	IF fbMoveAbsCA[0].Busy = FALSE THEN
		
		fbMoveAbsCA[0].Jerk			:= MotionParameters.Jerk;
		fbMoveAbsCA[0].Acceleration	:= MotionParameters.Acceleration;
		fbMoveAbsCA[0].Deceleration	:= MotionParameters.Deceleration;
		fbMoveAbsCA[0].Velocity		:= MotionParameters.Velocity;
		fbMoveAbsCA[0].Direction	:= MotionParameters.Direction;
		fbMoveAbsCA[0].Options.DynamicsReferenceSystem := CurrentTrack^.OTCID;
		fbMoveAbsCA[0].Options.PositionReferenceSystem := CurrentTrack^.OTCID;
		
		fbMoveAbsCA[0].Position		:= DestinationPosition;
		
		fbMoveAbsCA[0].BufferMode	:= mcAborting;
		fbMoveAbsCA[0].Execute		:= TRUE;
		 
		fbMoveAbsCA[0].Execute		:= TRUE;		// execute this block, and...
		fbMoveAbsCA[1].Execute		:= FALSE;		// if necessary, interrupt this one
		
		fbMoveAbsCA[0]( Axis := AxisReference );
		
	ELSIF fbMoveAbsCA[1].Busy = FALSE THEN
		
		fbMoveAbsCA[1].Jerk			:= MotionParameters.Jerk;
		fbMoveAbsCA[1].Acceleration	:= MotionParameters.Acceleration;
		fbMoveAbsCA[1].Deceleration	:= MotionParameters.Deceleration;
		fbMoveAbsCA[1].Velocity		:= MotionParameters.Velocity;
		fbMoveAbsCA[1].Direction	:= MotionParameters.Direction;
		fbMoveAbsCA[1].Options.DynamicsReferenceSystem := CurrentTrack^.OTCID;
		fbMoveAbsCA[1].Options.PositionReferenceSystem := CurrentTrack^.OTCID;

		
		fbMoveAbsCA[1].Position		:= DestinationPosition;
		
		fbMoveAbsCA[1].BufferMode	:= mcAborting;
		fbMoveAbsCA[1].Execute		:= TRUE;
		
		fbMoveAbsCA[1].Execute		:= TRUE;		// execute this block, and...
		fbMoveAbsCA[0].Execute		:= FALSE;		// if necessary, interrupt this one
		
		fbMoveAbsCA[1]( Axis := AxisReference );
		 
	ELSE
		MsgCreate.CreateEx( TC_EVENTS.XtsBaseEventClass.MoverMoveToPositionOverload,0 );
		MsgCreate.ipArguments.Clear().AddString(THIS^.InstancePath).AddString(THIS^.SourceInstancePath).AddLReal(DestinationPosition);
		MsgCreate.Send(0);
	END_IF
	
END_IF

internalCurrentMoveType		:= MOVETYPE_POSITION;
internalCurrentDestPosition := DestinationPosition;

memset( ADR( internalCurrentDestObjective ), 0, SIZEOF( internalCurrentDestObjective ));
internalCurrentDestStation	REF= 0;

IF ( newCallTime - lastCallMovePos ) > 1 THEN
	MsgCreate.CreateEx( TC_EVENTS.XtsBaseEventClass.MoverMoveToPosition,0 );
	MsgCreate.ipArguments.Clear().AddString(THIS^.InstancePath).AddString(THIS^.SourceInstancePath).AddLReal(DestinationPosition);
	MsgCreate.Send(0);
END_IF;

THIS^.SourceInstancePath	:= 'Direct access';

lastCallMovePos		:= newCallTime;

MoveToPosition		:= THIS^;
END_METHOD

METHOD MoveToStation : iMover
VAR_INPUT
	DestinationStation	: REFERENCE TO Station;	
END_VAR
VAR
	newCallTime			: LREAL;
END_VAR
VAR_INST
	MsgCreate			: FB_TcMessage;	
END_VAR
IF NOT( Ready ) AND NOT(__ISVALIDREF( DestinationStation )) THEN	// if the mover is not ready & able to accept a moveabs command...
	
	internalState	:= MV_ERROR;
	ErrorID			:= 19201;
	
ELSE	// otherwise let 'er rip
	
	newCallTime		:= ULINT_TO_LREAL(F_GetSystemTime())/1E7;
	internalReissue := FALSE;	// reissue no longer necessary
	
	IF fbMoveAbsCA[0].Busy = FALSE THEN
		
		fbMoveAbsCA[0].Jerk			:= MotionParameters.Jerk;
		fbMoveAbsCA[0].Acceleration	:= MotionParameters.Acceleration;
		fbMoveAbsCA[0].Deceleration	:= MotionParameters.Deceleration;
		fbMoveAbsCA[0].Velocity		:= MotionParameters.Velocity;
		fbMoveAbsCA[0].Direction	:= MotionParameters.Direction;
		fbMoveAbsCA[0].Options.DynamicsReferenceSystem := CurrentTrack^.OTCID;
		fbMoveAbsCA[0].Options.PositionReferenceSystem := CurrentTrack^.OTCID;
		
		fbMoveAbsCA[0].Position		:= DestinationStation.internalPosition;
		
		fbMoveAbsCA[0].BufferMode	:= mcAborting;
		fbMoveAbsCA[0].Execute		:= TRUE;
		 
		fbMoveAbsCA[0].Execute		:= TRUE;		// execute this block, and...
		fbMoveAbsCA[1].Execute		:= FALSE;		// if necessary, interrupt this one
		
		fbMoveAbsCA[0]( Axis := AxisReference );
		
	ELSIF fbMoveAbsCA[1].Busy = FALSE THEN
		
		fbMoveAbsCA[1].Jerk			:= MotionParameters.Jerk;
		fbMoveAbsCA[1].Acceleration	:= MotionParameters.Acceleration;
		fbMoveAbsCA[1].Deceleration	:= MotionParameters.Deceleration;
		fbMoveAbsCA[1].Velocity		:= MotionParameters.Velocity;
		fbMoveAbsCA[1].Direction	:= MotionParameters.Direction;
		fbMoveAbsCA[1].Options.DynamicsReferenceSystem := CurrentTrack^.OTCID;
		fbMoveAbsCA[1].Options.PositionReferenceSystem := CurrentTrack^.OTCID;
		
		fbMoveAbsCA[1].Position		:= DestinationStation.internalPosition;
		
		fbMoveAbsCA[1].BufferMode	:= mcAborting;
		fbMoveAbsCA[1].Execute		:= TRUE;
		
		fbMoveAbsCA[1].Execute		:= TRUE;		// execute this block, and...
		fbMoveAbsCA[0].Execute		:= FALSE;		// if necessary, interrupt this one

		fbMoveAbsCA[1]( Axis := AxisReference );	

	ELSE
		MsgCreate.CreateEx( TC_EVENTS.XtsBaseEventClass.MoverMoveToStationOverload,0 );
		MsgCreate.ipArguments.Clear().AddString(THIS^.InstancePath).AddString(THIS^.SourceInstancePath).AddString(DestinationStation.InstancePath);
		MsgCreate.Send(0);
		
	END_IF
	
	// Set the current destination object to the instance path of the objective, or 0 if unassigned
	internalCurrentDestPosition		:= DestinationStation.Position;
	internalCurrentDestObjective	:= SEL( __ISVALIDREF( DestinationStation ), '', DestinationStation.InstancePath );
	internalCurrentDestStation		REF= DestinationStation;
	internalCurrentMoveType			:= MOVETYPE_STATION;
	
	// Register this mover with the station, so the station knows this mover is incoming
	DestinationStation.RegisterMover( THIS^ );
	
END_IF

IF ( newCallTime - lastCallMoveSta ) > 1 THEN
	MsgCreate.CreateEx( TC_EVENTS.XtsBaseEventClass.MoverMoveToStation,0 );
	MsgCreate.ipArguments.Clear().AddString(THIS^.InstancePath).AddString(THIS^.SourceInstancePath).AddString(DestinationStation.InstancePath);
	MsgCreate.Send(0);
END_IF

THIS^.SourceInstancePath	:= 'Direct access';

lastCallMoveSta		:= newCallTime;

MoveToStation		:= THIS^;
END_METHOD

METHOD MoveVelocity : iMover
VAR_INPUT
	DesiredVelocity : LREAL;		//The velocity to be commanded [mm/s]
END_VAR
VAR
	negativeCommand	: BOOL;
	newCallTime		: LREAL;
END_VAR
VAR_INST
	MsgCreate		: FB_TcMessage;	
END_VAR
IF NOT ( ready ) THEN
	
	internalState	:= MV_ERROR;
	ErrorID			:= 19201;
	
ELSE
	
	newCallTime		:= ULINT_TO_LREAL(F_GetSystemTime())/1E7;
	internalReissue := FALSE;	// reissue no longer necessary
	
	negativeCommand					:= SEL( DesiredVelocity < 0, FALSE, TRUE );
	MotionParameters.Velocity		:= ABS( DesiredVelocity );
	
	IF fbMoveRelCA[0].Busy = FALSE THEN
		
		fbMoveRelCA[0].Jerk			:= MotionParameters.Jerk;
		
		fbMoveRelCA[0].Acceleration	:= MotionParameters.Acceleration;
		fbMoveRelCA[0].Deceleration	:= MotionParameters.Deceleration;
		fbMoveRelCA[0].Velocity		:= MotionParameters.Velocity;
		
		fbMoveRelCA[0].Distance		:= SEL( negativeCommand, 1E100, -1E100 );
		
		      
		fbMoveRelCA[0].BufferMode	:= mcAborting;
		      
		fbMoveRelCA[0].Execute		:= TRUE;		// execute this block, and...
		fbMoveRelCA[1].Execute		:= FALSE;		// if necessary, interrupt this one
		
		fbMoveRelCA[0]( Axis := AxisReference );
		
	ELSIF fbMoveRelCA[1].Busy = FALSE THEN
		
		fbMoveRelCA[1].Jerk			:= MotionParameters.Jerk;
		
		fbMoveRelCA[1].Acceleration	:= MotionParameters.Acceleration;
		fbMoveRelCA[1].Deceleration	:= MotionParameters.Deceleration;
		fbMoveRelCA[1].Velocity		:= MotionParameters.Velocity;
		      
		fbMoveRelCA[1].Distance		:= SEL( negativeCommand, 1E100, -1E100 );
		      
		fbMoveRelCA[1].BufferMode	:= mcAborting;
		      
		fbMoveRelCA[1].Execute		:= TRUE;		// execute this block, and...
		fbMoveRelCA[0].Execute		:= FALSE;		// if necessary, interrupt this one

		fbMoveRelCA[1]( Axis := AxisReference );
	ELSE
		MsgCreate.CreateEx( TC_EVENTS.XtsBaseEventClass.MoverMoveVelocityOverload,0 );
		MsgCreate.ipArguments.Clear().AddString(THIS^.InstancePath).AddString(THIS^.SourceInstancePath).AddLReal(DesiredVelocity);
		MsgCreate.Send(0);
	END_IF

END_IF

fbMoveRelCA[0] ( Axis := AxisReference );
fbMoveRelCA[1] ( Axis := AxisReference );


internalCurrentMoveType		:= MOVETYPE_VELOCITY;
internalCurrentDestPosition := 1E300;

memset( ADR( internalCurrentDestObjective ), 0, SIZEOF( internalCurrentDestObjective ));
internalCurrentDestStation	REF= 0;

IF ( newCallTime - lastCallMoveVel ) > 1 THEN
	MsgCreate.CreateEx( TC_EVENTS.XtsBaseEventClass.MoverMoveVelocity,0 );
	MsgCreate.ipArguments.Clear().AddString(THIS^.InstancePath).AddString(THIS^.SourceInstancePath).AddLReal(DesiredVelocity);
	MsgCreate.Send(0);
END_IF;

THIS^.SourceInstancePath	:= 'Direct access';

lastCallMoveVel		:= newCallTime;

MoveVelocity		:= THIS^;
END_METHOD

PROPERTY Payload : Payload_typ
GET


Payload	:= internalPayload;
END_GET
SET


internalPayload	:= Payload;
END_SET
END_PROPERTY

METHOD ReissueCommand : iMover
VAR_INPUT
END_VAR

// set flag for use in .Cyclic()
internalReissue := TRUE;


ReissueCommand		:= THIS^;
END_METHOD

METHOD SetAcceleration : iMover
VAR_INPUT
	Acceleration	: LREAL;
END_VAR
VAR
	newCallTime		: LREAL;
END_VAR
VAR_INST
	MsgCreate		: FB_TcMessage;	
END_VAR

newCallTime		:= ULINT_TO_LREAL(F_GetSystemTime())/1E7;

MotionParameters.Acceleration		:= LIMIT( 0, Acceleration, 1E300 );	// upper limit is capped by the axis object parameters

THIS^.ReissueCommand();

IF ( newCallTime - lastCallSetAcc ) > 1 THEN
	MsgCreate.CreateEx( TC_EVENTS.XtsBaseEventClass.MoverSetAcceleration,0 );
	MsgCreate.ipArguments.Clear().AddString(THIS^.InstancePath).AddString(THIS^.SourceInstancePath).AddLReal(Acceleration);
	MsgCreate.Send(0);
END_IF;

THIS^.SourceInstancePath	:= 'Direct access';

lastCallSetAcc		:= newCallTime;

SetAcceleration		:= THIS^;
END_METHOD

METHOD SetDeceleration : iMover
VAR_INPUT
	Deceleration	: LREAL;
END_VAR
VAR
	newCallTime		: LREAL;
END_VAR
VAR_INST
	MsgCreate		: FB_TcMessage;	
END_VAR

newCallTime		:= ULINT_TO_LREAL(F_GetSystemTime())/1E7;

MotionParameters.Deceleration	:= LIMIT( 0, Deceleration, 1E300 ); // upper limit is capped by the axis parameters

THIS^.ReissueCommand();

IF ( newCallTime - lastCallSetDec ) > 1 THEN
	MsgCreate.CreateEx( TC_EVENTS.XtsBaseEventClass.MoverSetDeceleration,0 );
	MsgCreate.ipArguments.Clear().AddString(THIS^.InstancePath).AddString(THIS^.SourceInstancePath).AddLReal(Deceleration);
	MsgCreate.Send(0);
END_IF

THIS^.SourceInstancePath	:= 'Direct access';

lastCallSetDec		:= newCallTime;

SetDeceleration		:= THIS^;
END_METHOD

METHOD SetDirection : iMover
VAR_INPUT
	Direction		: Tc3_Mc3Definitions.MC_Direction;
END_VAR
VAR
	newCallTime		: LREAL;
END_VAR
VAR_INST
	MsgCreate		: FB_TcMessage;	
END_VAR

newCallTime		:= ULINT_TO_LREAL(F_GetSystemTime())/1E7;

MotionParameters.Direction		:= Direction;

THIS^.ReissueCommand();

IF ( newCallTime - lastCallSetDir ) > 1 THEN
	MsgCreate.CreateEx( TC_EVENTS.XtsBaseEventClass.MoverSetDirection,0 );
	MsgCreate.ipArguments.Clear().AddString(THIS^.InstancePath).AddString(THIS^.SourceInstancePath).AddInt(Direction);
	MsgCreate.Send(0);
END_IF

THIS^.SourceInstancePath	:= 'Direct access';

lastCallSetDir		:= newCallTime;

SetDirection		:= THIS^;
END_METHOD

METHOD SetJerk : iMover
VAR_INPUT
	Jerk		: LREAL;
END_VAR
VAR
	newCallTime	: LREAL;
END_VAR
VAR_INST
	MsgCreate	: FB_TcMessage;	
END_VAR

newCallTime		:= ULINT_TO_LREAL(F_GetSystemTime())/1E7;

MotionParameters.Jerk		:= LIMIT( 0, Jerk, 1E300 ); // upper limit is capped by the axis parameters

THIS^.ReissueCommand();

IF ( newCallTime - lastCallSetJerk ) > 1 THEN
	MsgCreate.CreateEx( TC_EVENTS.XtsBaseEventClass.MoverSetJerk,0 );
	MsgCreate.ipArguments.Clear().AddString(THIS^.InstancePath).AddString(THIS^.SourceInstancePath).AddLReal(Jerk);
	MsgCreate.Send(0);
END_IF

THIS^.SourceInstancePath	:= 'Direct access';

lastCallSetJerk		:= newCallTIme;

SetJerk		:= THIS^;
END_METHOD

METHOD SetVelocity : iMover
VAR_INPUT
	Velocity		: LREAL;		// Updates Mover's internal velocity parameter. Takes effect immediately. [mm/s]
END_VAR
VAR
	logstr			: STRING(200);		// method variable containing an event log message for the command
	LogEvent		: INT;
	newCallTime		: LREAL;
END_VAR
VAR_INST
	MsgCreate		: FB_TcMessage;	
END_VAR

newCallTime		:= ULINT_TO_LREAL(F_GetSystemTime())/1E7;

MotionParameters.Velocity	:= LIMIT( 0, Velocity, 1E300 ); // upper limit is capped by the axis parameters 

THIS^.ReissueCommand();

IF ( newCallTime - lastCallSetVel ) > 1 THEN
	MsgCreate.CreateEx( TC_EVENTS.XtsBaseEventClass.MoverSetVelocity,0 );
	MsgCreate.ipArguments.Clear().AddString(THIS^.InstancePath).AddString(THIS^.SourceInstancePath).AddLReal(Velocity);
	MsgCreate.Send(0);
END_IF

THIS^.SourceInstancePath	:= 'Direct access';

lastCallSetVel	:= newCallTime;

SetVelocity		:= THIS^;
END_METHOD

METHOD SyncToAxis : iMover
VAR_INPUT
	
	MasterAxis		: REFERENCE TO AXIS_REF;
	MasterSyncPos	: LREAL;				// Master sync position (nonmodulo), where the input axis will be located when first synchronized
	SlaveSyncPos	: LREAL;				// Mover sync position, where the mover will be located when first synchronized
	SyncStrategy	: MC_SYNC_STRATEGY;		// Direction input
	
END_VAR
VAR
	newCallTime		: LREAL;
END_VAR
VAR_INST
	MsgCreate		: FB_TcMessage;
END_VAR


IF NOT( Ready ) THEN
	
	internalState		:= MV_ERROR;
	ErrorID				:= 19201;
	
ELSE
	
	newCallTime			:= ULINT_TO_LREAL(F_GetSystemTime())/1E7;
	internalReissue := FALSE;	// reissue no longer necessary
	
	internalMasterAxis		REF= MasterAxis;
	
	IF fbGearInPosAxisCA[0].Busy = FALSE THEN
		
		fbGearInPosAxisCA[0].Execute			:= TRUE;
		
		fbGearInPosAxisCA[0].RatioNumerator		:= 1;
		fbGearInPosAxisCA[0].RatioDenumerator	:= 1;
		
		fbGearInPosAxisCA[0].MasterSyncPosition	:= MasterSyncPos;	// This needs to be nonmodulo
		fbGearInPosAxisCA[0].SlaveSyncPosition	:= SlaveSyncPos;
		
		fbGearInPosAxisCA[0].SyncStrategy		:= SyncStrategy;
		
		fbGearInPosAxisCA[0].Options.DynamicsReferenceSystem := CurrentTrack^.OTCID;
		fbGearInPosAxisCA[0].Options.SlaveSyncPositionReferenceSystem := CurrentTrack^.OTCID;

		
		IF MotionParameters.Direction = mcDirectionPositive THEN
			fbGearInPosAxisCA[0].SyncMode		:= mcSyncModePositive;
		ELSIF MotionParameters.Direction = mcDirectionNegative THEN
			fbGearInPosAxisCA[0].SyncMode		:= mcSyncModeNegative;
		END_IF
		
		fbGearInPosAxisCA[0].Velocity			:= MotionParameters.Velocity;
		fbGearInPosAxisCA[0].Acceleration		:= MotionParameters.Acceleration;
		fbGearInPosAxisCA[0].Deceleration		:= MotionParameters.Deceleration;
		fbGearInPosAxisCA[0].Jerk				:= MotionParameters.Jerk;
		
		fbGearInPosAxisCA[0].BufferMode			:= Tc3_Mc3Definitions.MC_BUFFER_MODE.mcAborting;
		
		fbGearInPosAxisCA[0]( Master := MasterAxis, Slave := THIS^.AxisReference );		
		
	ELSIF fbGearInPosAxisCA[1].Busy = FALSE THEN
		
		fbGearInPosAxisCA[1].Execute			:= TRUE;
		
		fbGearInPosAxisCA[1].RatioNumerator		:= 1;
		fbGearInPosAxisCA[1].RatioDenumerator	:= 1;
		
		fbGearInPosAxisCA[1].MasterSyncPosition	:= MasterSyncPos;	// This needs to be nonmodulo
		fbGearInPosAxisCA[1].SlaveSyncPosition	:= SlaveSyncPos;
		
		fbGearInPosAxisCA[1].SyncStrategy		:= SyncStrategy;
		
		fbGearInPosAxisCA[1].Options.DynamicsReferenceSystem := CurrentTrack^.OTCID;
		fbGearInPosAxisCA[1].Options.SlaveSyncPositionReferenceSystem := CurrentTrack^.OTCID;
		
		IF MotionParameters.Direction = mcDirectionPositive THEN
			fbGearInPosAxisCA[1].SyncMode		:= mcSyncModePositive;
		ELSIF MotionParameters.Direction = mcDirectionNegative THEN
			fbGearInPosAxisCA[1].SyncMode		:= mcSyncModeNegative;				
		END_IF
		
		fbGearInPosAxisCA[1].Velocity			:= MotionParameters.Velocity;
		fbGearInPosAxisCA[1].Acceleration		:= MotionParameters.Acceleration;
		fbGearInPosAxisCA[1].Deceleration		:= MotionParameters.Deceleration;
		fbGearInPosAxisCA[1].Jerk				:= MotionParameters.Jerk;
		
		fbGearInPosAxisCA[1].BufferMode			:= Tc3_Mc3Definitions.MC_BUFFER_MODE.mcAborting;
		
		fbGearInPosAxisCA[1]( Master := MasterAxis, Slave := THIS^.AxisReference );

	ELSE
		MsgCreate.CreateEx( TC_EVENTS.XtsBaseEventClass.MoverSyncToAxisOverload, 0 );
		MsgCreate.ipArguments.Clear().AddString(THIS^.InstancePath).AddString(THIS^.SourceInstancePath);
		MsgCreate.Send(0);
	END_IF
	
END_IF

internalCurrentMoveType			:= MOVETYPE_SYNC_AXIS;
internalCurrentDestPosition		:= 1E300;

memset( ADR( internalCurrentDestObjective ), 0, SIZEOF( internalCurrentDestObjective ));
internalCurrentDestStation		REF= 0;

IF ( newCallTime - lastCallSync ) > 1 THEN
	MsgCreate.CreateEx( TC_EVENTS.XtsBaseEventClass.MoverSyncToAxis, 0 );
	MsgCreate.ipArguments.Clear().AddString(THIS^.InstancePath).AddString(THIS^.SourceInstancePath);
	MsgCreate.Send(0);
END_IF

THIS^.SourceInstancePath		:= 'Direct access';

lastCallSync	:= newCallTime;

SyncToAxis		:= THIS^;
END_METHOD

METHOD SyncToMover : iMover
VAR_INPUT
	MasterMover			: REFERENCE TO Mover;	// Synchronization master mover, whose position to follow. Further motion commands break the pairing
	Gap					: LREAL;				// Gap distance to lead mover. Positive values indicate following, negative values indicate leading
END_VAR
VAR
	CWDistToSync		: LREAL;
	CWDistToMaster		: LREAL;
	syncPos				: LREAL;
	newCallTime			: LREAL;
END_VAR
VAR_INST
	MsgCreate			: FB_TcMessage;	
END_VAR
IF NOT( Ready ) THEN

	internalState	:= MV_ERROR;
	ErrorID			:= 19201;
	
ELSE	// let 'er rip
	
	newCallTime		:= ULINT_TO_LREAL(F_GetSystemTime())/1E7;
	internalReissue := FALSE;	// reissue no longer necessary

	internalMasterMover		REF= MasterMover;
	internalGap				:= Gap;
	
	
	syncPos			:= internalMasterMover.AxisReference.NcToPlc.ActPos - internalGap;
	CWDistToSync	:= MODABS( syncPos - THIS^.AxisReference.NcToPlc.ActPos, GVL.TRACK_LENGTH );
	CWDistToMaster	:= MODABS( internalMasterMover.AxisReference.NcToPlc.ActPos - THIS^.AxisReference.NcToPlc.ActPos, GVL.TRACK_LENGTH );
		
	IF fbGearInPosMoverCA[0].Busy = FALSE THEN
		
		fbGearInPosMoverCA[0].Execute				:= TRUE;
			
		fbGearInPosMoverCA[0].RatioNumerator			:= 1;
		fbGearInPosMoverCA[0].RatioDenumerator		:= 1;
		
		fbGearInPosMoverCA[0].MasterSyncPosition		:= internalMasterMover.AxisReference.NcToPlc.ActPos;
		fbGearInPosMoverCA[0].SlaveSyncPosition		:= MODABS( internalMasterMover.AxisReference.NcToPlc.ActPos - internalGap, GVL.TRACK_LENGTH);
		
		fbGearInPosMoverCA[0].SyncStrategy			:= mcSyncStrategyEarly;		
		fbGearInPosMoverCA[0].SyncMode				:= SEL( CWDistToSync < CWDistToMaster, mcSyncModeNegative, mcSyncModePositive );
				
		//fbGearInPosMoverCA[0].Options.MinimalSlavePosition	:= -1E300;
		
		fbGearInPosMoverCA[0].Velocity				:= MotionParameters.Velocity;
		fbGearInPosMoverCA[0].Acceleration			:= MotionParameters.Acceleration;
		fbGearInPosMoverCA[0].Deceleration			:= MotionParameters.Deceleration;
		fbGearInPosMoverCA[0].Jerk					:= MotionParameters.Jerk;
		
		fbGearInPosMoverCA[0].BufferMode				:= Tc3_Mc3Definitions.MC_BUFFER_MODE.mcAborting;
		
		fbGearInPosMoverCA[0]( Master := internalMasterMover.AxisReference, Slave := THIS^.AxisReference );
		
	ELSIF fbGearInPosMoverCA[1].Busy = FALSE THEN
		
		fbGearInPosMoverCA[1].Execute				:= TRUE;
		
		fbGearInPosMoverCA[1].RatioNumerator			:= 1;
		fbGearInPosMoverCA[1].RatioDenumerator		:= 1;
		
		fbGearInPosMoverCA[1].MasterSyncPosition		:= internalMasterMover.AxisReference.NcToPlc.ActPos;
		fbGearInPosMoverCA[1].SlaveSyncPosition		:= MODABS( internalMasterMover.AxisReference.NcToPlc.ActPos - internalGap, GVL.TRACK_LENGTH);
		
		fbGearInPosMoverCA[1].SyncStrategy			:= mcSyncStrategyEarly;
		fbGearInPosMoverCA[1].SyncMode				:= SEL( CWDistToSync < CWDistToMaster, mcSyncModeNegative, mcSyncModePositive );
		
		//fbGearInPosMoverCA[1].Options.MinimalSlavePosition	:= -1E300;
		
		fbGearInPosMoverCA[1].Velocity				:= MotionParameters.Velocity;
		fbGearInPosMoverCA[1].Acceleration			:= MotionParameters.Acceleration;
		fbGearInPosMoverCA[1].Deceleration			:= MotionParameters.Deceleration;
		fbGearInPosMoverCA[1].Jerk					:= MotionParameters.Jerk;
		
		fbGearInPosMoverCA[1].BufferMode				:= Tc3_Mc3Definitions.MC_BUFFER_MODE.mcAborting;
		
		
		fbGearInPosMoverCA[1]( Master := internalMasterMover.AxisReference, Slave := THIS^.AxisReference );
		
	ELSE
		MsgCreate.CreateEx( TC_EVENTS.XtsBaseEventClass.MoverSyncToMoverOverload,0 );
		MsgCreate.ipArguments.Clear().AddString(THIS^.InstancePath).AddString(THIS^.SourceInstancePath).AddString(MasterMover.InstancePath).AddLReal(Gap);
		MsgCreate.Send(0);
		
	END_IF

END_IF;

internalCurrentMoveType			:= MOVETYPE_SYNC_MOVER;
internalCurrentDestPosition		:= 1E300;

memset( ADR( internalCurrentDestObjective ), 0, SIZEOF( internalCurrentDestObjective ));
internalCurrentDestStation	REF= 0;

IF ( newCallTime - lastCallSync ) > 1 THEN
	MsgCreate.CreateEx( TC_EVENTS.XtsBaseEventClass.MoverSyncToMover,0 );
	MsgCreate.ipArguments.Clear().AddString(THIS^.InstancePath).AddString(THIS^.SourceInstancePath).AddString(MasterMover.InstancePath).AddLReal(Gap);
	MsgCreate.Send(0);
END_IF

THIS^.SourceInstancePath	:= 'Direct access';

lastCallSync		:= newCallTime;


SyncToMover		:= THIS^;
END_METHOD

END_FUNCTION_BLOCK

(* stored: Version 1.1.0.1, ProductVersion 3.1.4024.12
   POU Mover: Id {461a92b9-026e-4cbb-aa50-b18297f25ecc}, SpecialFunc None
   Folder Methods: Id {d146b766-1176-40b7-a641-ffa579406c77}
   Folder Properties: Id {9b9301bf-13c1-4ce0-91ab-e61950dfd74a}
   Method ActivateTrack: Id {2cd7eff7-09ea-0845-346b-196f53ea2e60}
   Property CurrentDestinationPosition: Id {6d470b15-bd31-4ad6-8559-906c2c8d720c}
   Get Get: Id {bc93c9f7-92a5-426e-9c7f-5953d1b7c034}
   Property CurrentMoveType: Id {97c82f4e-fad3-4ecf-8f48-6f47f3a34a61}
   Get Get: Id {008a2288-6099-47d9-88ab-640a99950162}
   Property CurrentObjective: Id {b06cf2ff-b1dd-4afb-af24-76820a9809f8}
   Get Get: Id {39f22891-e1d0-4fbf-9032-2bbc45b18310}
   Property CurrentTrack: Id {57746913-d241-0290-0366-208479410de1}
   Get Get: Id {845db4a8-12f5-01df-23b2-2ce5c8663c6a}
   Method Cyclic: Id {39769063-232f-402c-8c9b-ad47db196752}
   Method CyclicTrack: Id {f91ef8d2-f744-0809-3990-5a057546bb09}
   Method Disable: Id {2aa14795-54cd-46b8-a131-b1a8801c005f}
   Method Enable: Id {77bc5ebc-ace3-48eb-8e85-e45bc80ac98b}
   Method GroupStop: Id {19a65925-9b39-4de9-ab16-7733d66c5fd4}
   Method Halt: Id {1f55ad78-11ad-492d-9f7a-e48ae6feda84}
   Property IsSyncedToAxis: Id {f2757d0f-8cc6-01d8-3ce1-c233354ecef8}
   Get Get: Id {1582f1e6-442b-0b9d-21b6-52b967b5912b}
   Property IsSyncedToMover: Id {b02e7e76-e41b-42cd-ad2a-fd14e80d7543}
   Get Get: Id {b38e44ed-4371-4ccd-ba7f-e98ea73ca608}
   Property IsTrackReady: Id {cd5c6866-73e3-00ad-2292-5fe936355763}
   Get Get: Id {1b14d83a-1ec1-0d2f-1616-ce7f9ce5cce5}
   Method LogUserEvent: Id {2ade5417-e15a-4da8-a731-8eb7341e5999}
   Property MasterMover: Id {809c0b0b-ecf0-4af1-b9a6-f6c1668f1e51}
   Get Get: Id {cf9c37de-0f5d-4ab8-bb6c-0c7a9a276e2e}
   Method MoveToMultiStation: Id {ae99d1c6-e395-0e0a-0cfd-93b12a0892ad}
   Method MoveToPosition: Id {c28d081f-5f21-4357-8651-768a8cf4ef0e}
   Method MoveToStation: Id {73370b80-491c-4017-a420-f08c462d830e}
   Method MoveVelocity: Id {b843a8f8-3644-434c-aaf5-7e88053f31b1}
   Property Payload: Id {5caf95a6-ad6c-448d-8947-8c8c07ab0a26}
   Get Get: Id {8a73f5fd-2b02-4094-9725-10c35f9f9334}
   Set Set: Id {6f8bbb61-047b-455a-a948-12da14d2f890}
   Method ReissueCommand: Id {195ecbe2-3d92-4d60-b9b5-7e1a3292ea5b}
   Method SetAcceleration: Id {6c3e67ff-faff-4c11-8768-1de83c7995e4}
   Method SetDeceleration: Id {05a8542e-78cf-4f19-864b-98da64430703}
   Method SetDirection: Id {e0c3c5b2-5259-4ab4-9ff7-1ecaf9015b31}
   Method SetJerk: Id {de57e13f-25de-42a4-aec6-c6dc8b78d964}
   Method SetVelocity: Id {530483ab-165f-437b-baf5-2db027b7f044}
   Method SyncToAxis: Id {6776bdec-2c5f-03ab-27c8-402842cfde2e}
   Method SyncToMover: Id {c1dddc96-f9c0-4f4e-b1ac-4bb8d23d72f1} *)
